Yaskawa INFORM job: FMTV_HOOD_LEFT.JBI

/JOB
//NAME FMTV_HOOD_LEFT
//POS
///NPOS 70,0,0,0,0,0
///TOOL 0
///POSTYPE PULSE
///PULSE
C00000=-252640,-156391,-84960,58658,-32345,33822
C00001=-156384,-125973,-74844,178526,55936,-172151
C00002=-135851,-173202,-20342,60003,118037,36627
C00003=-128704,-166266,35271,81917,119544,44528
C00004=-128536,-164580,41005,80917,119261,43270
C00005=-129375,-164845,40778,80344,119100,43271
C00006=-129497,-164201,41559,80229,119066,43235
C00007=-126845,-168006,35684,82558,119695,32854
C00008=-126480,-161319,43205,86363,112864,32361
C00009=-126433,-157348,47941,88535,108968,31899
C00010=-126470,-154595,51339,90015,106365,31512
C00011=-126409,-156094,57474,97995,109328,16701
C00012=-126708,-159160,48051,98861,108825,18520
C00013=-127111,-159008,46055,100189,106138,23442
C00014=-130033,-155814,41530,96820,92589,41961
C00015=-152223,-172084,23477,70836,100058,41015
C00016=-152223,-172084,23477,70836,100058,41015
C00017=-152648,-172193,23550,70529,99976,40976
C00018=-153063,-171996,23911,70229,99900,40943
C00019=-153497,-170611,31323,73841,101293,23588
C00020=-154147,-171465,28414,73593,101484,24157
C00021=-157584,-164927,35202,71230,100976,24221
C00022=-154632,-160160,47280,75419,109863,8591
C00023=-154632,-160160,47280,75419,109863,8591
C00024=-155625,-160292,45598,75022,109882,9061
C00025=-156123,-160064,44186,74976,110013,9541
C00026=-156123,-160064,44186,74976,110013,9541
C00027=-156123,-160064,44186,74976,110013,9541
C00028=-156487,-159930,43303,74905,110090,9841
C00029=-157445,-159958,41921,74498,110121,10251
C00030=-158548,-160172,40798,73908,110078,10536
C00031=-159546,-160463,40026,73314,109996,10697
C00032=-159546,-160463,40026,73314,109996,10697
C00033=-159546,-160463,40026,73314,109996,10697
C00034=-160288,-160677,39489,72866,109936,10807
C00035=-161356,-160813,38506,72286,109910,11066
C00036=-161512,-160713,38768,72381,111191,8601
C00037=-161088,-159950,39557,72687,115021,1476
C00038=-159810,-165209,31993,74041,115511,2080
C00039=-158925,-166012,40140,122202,116650,-14944
C00040=-160518,-162642,45165,133205,115264,-20836
C00041=-119253,-154583,37644,271020,100127,-40659
C00042=-117173,-142082,66967,267962,96812,-36379
C00043=-116899,-137930,76717,268472,96896,-34848
C00044=-122642,-140335,66800,272097,94183,-36590
C00045=-122642,-140335,66800,272097,94183,-36590
C00046=-123853,-142202,60931,276553,92212,-37524
C00047=-126842,-142231,60643,274488,92717,-37576
C00048=-126842,-142231,60643,274488,92717,-37576
C00049=-126842,-142231,60643,274488,92717,-37576
C00050=-127969,-142503,60272,273708,92904,-37597
C00051=-129474,-143238,59510,272670,93154,-37596
C00052=-130457,-143972,58745,271991,93315,-37600
C00053=-130457,-143972,58745,271991,93315,-37600
C00054=-130457,-143972,58745,271991,93315,-37600
C00055=-132216,-144423,58503,271361,94455,-38217
C00056=-135829,-145042,58868,269290,97087,-39237
C00057=-138484,-145389,59559,267670,99169,-39937
C00058=-139384,-145389,60026,267056,99942,-40165
C00059=-140047,-145511,60188,266706,100449,-40337
C00060=-141803,-145775,60748,265711,101855,-40793
C00061=-143397,-145936,61441,264719,103223,-41200
C00062=-143962,-146001,61697,264342,103732,-41344
C00063=-148001,-148124,61021,263058,107890,-40745
C00064=-151541,-150083,60557,262198,111774,-40091
C00065=-153305,-151022,60467,261910,113836,-39700
C00066=-159207,-156478,57346,261381,118432,-38208
C00067=-165627,-162538,55030,261269,123130,-36160
C00068=-166488,-164984,48680,259443,122976,-37429
C00069=-147066,-165395,-6439,251998,122776,-36821
//INST
///DATE 2022/03/25 15:05
///ATTR SC,RW
///GROUP1 RB1
NOP
MOVJ C00000 VJ=65.00  //FROM FLASH
MOVJ C00001 VJ=65.00
MOVJ C00002 VJ=65.00
MOVL C00003 V=65.0  //UP TO
MOVL C00004 V=15.0  //INTO
MOVL C00005 V=15.0
MOVL C00006 V=15.0
MOVL C00007 V=15.0
MOVL C00008 V=15.0
MOVL C00009 V=15.0
MOVL C00010 V=15.0
MOVL C00011 V=15.0
MOVL C00012 V=15.0
MOVL C00013 V=15.0
MOVL C00014 V=15.0
MOVL C00015 V=15.0
MOVC C00016 V=15.0
MOVC C00017 V=15.0
MOVC C00018 V=15.0
MOVL C00019 V=8.0
MOVL C00020 V=15.0
MOVL C00021 V=15.0
MOVL C00022 V=8.0
MOVC C00023 V=15.0
MOVC C00024 V=15.0
MOVC C00025 V=15.0
MOVL C00026 V=15.0
MOVC C00027 V=15.0
MOVC C00028 V=15.0
MOVC C00029 V=15.0
MOVC C00030 V=15.0
MOVC C00031 V=15.0
MOVL C00032 V=15.0
MOVC C00033 V=15.0
MOVC C00034 V=15.0
MOVC C00035 V=15.0
MOVL C00036 V=15.0
MOVL C00037 V=8.0  //END
MOVL C00038 V=45.0  //OUT
MOVL C00039 V=65.0
MOVL C00040 V=65.0
MOVL C00041 V=65.0
MOVL C00042 V=65.0  //UP TO BACK
MOVL C00043 V=15.0  //INTO BACK
MOVL C00044 V=15.0  //COMMENT
MOVC C00045 V=15.0
MOVC C00046 V=15.0
MOVC C00047 V=15.0
MOVL C00048 V=15.0
MOVC C00049 V=15.0
MOVC C00050 V=15.0
MOVC C00051 V=15.0
MOVC C00052 V=15.0
MOVL C00053 V=15.0
MOVC C00054 V=15.0
MOVC C00055 V=15.0
MOVC C00056 V=15.0
MOVC C00057 V=15.0
MOVC C00058 V=15.0
MOVC C00059 V=15.0
MOVC C00060 V=15.0
MOVC C00061 V=15.0
MOVC C00062 V=15.0
MOVC C00063 V=15.0
MOVC C00064 V=15.0
MOVC C00065 V=15.0
MOVC C00066 V=15.0
MOVC C00067 V=15.0
MOVL C00068 V=45.0  //OUT
MOVJ C00069 VJ=65.00
END
